PROGRAM Prg_Persistance
VAR
FB_S_UPS_CX8190	: FB_S_UPS_CX81xx;

END_VAR

FB_S_UPS_CX8190(	sNetID :='',
					iPLCPort        := 851, (* PLC Runtime System for writing persistent data *)
  					tTimeout        := DEFAULT_ADS_TIMEOUT, (* ADS Timeout *)
    				eUpsMode        := eSUPS_WrPersistData_Shutdown, (* UPS mode (w/wo writing persistent data, w/wo NO shutdown) *)
   					ePersistentMode := SPDM_2PASS, (* mode for writing persistent data *)
    				tRecoverTime    := T#10S, (* ON time to recover from short power failure in mode eSUPS_WrPersistData_NoShutdown/eSUPS_CheckPowerStatus *)
					);

END_PROGRAM

(* stored: Version 1.1.0.1, ProductVersion 3.1.4024.12
   POU Prg_Persistance: Id {ad865142-7ab1-4ee4-9c9b-55f1fdeb4d9f}, SpecialFunc None *)
